PROGRAM MAIN
VAR
END_VAR

POU();

END_PROGRAM

(* stored: Version 1.1.0.1, ProductVersion 3.1.4022.7
   POU MAIN: Id {d829f270-b452-495c-83eb-48e756c78ec4}, SpecialFunc None *)
